{attribute 'qualified_only'}
{attribute 'strict'}
TYPE eSetPositionMode :
(
    Absolute := 0,
    Relative := 1
);
END_TYPE

(* stored: Version 1.1.0.1, ProductVersion 3.1.4024.6
   DUT eSetPositionMode: Id {c73fdd70-cdaa-0b16-2d39-943a01c717ca} *)
